FUNCTION_BLOCK XtsHardware_TestSuite
VAR
	nullHardware : XTSHardware('');
	MyXtsHardware : XTSHardware('') := (ExpectedNumberOfParts := 1, ExpectedNumberOfTracks := 1);
	localXpu: Xts_Library.I_TcIoXtsProcessingUnit;
	ThisTestSuite : TestSuite<TestSuiteParameter.MaxTestCount>('C:\ProgramData\Beckhoff\TwinCAT\3.1\Boot\XtsHardware_Tests.xml') := (TestSuiteName := 'XtsHardware Test Suite');
END_VAR

IF NOT MyXtsHardware.Initialised THEN
	MyXtsHardware.Initialise();
	RETURN;
END_IF

HardwareAcceptsTrackForDetection_Test();
HardwareAcceptsValidGetTrack_Test();
HardwareRejectsOnlyTrackRemove_Test();
HardwareIdentifiesNoXpu_Test();
HardwareRejectsCallsWithNoXPU_Test();
HardwareRejectsGetTrackWithHighTrackNum_Test();
HardwareRejectsGetTrackWithNull_Test();
HardwareRejectsHighIndexTrackRemoval_Test();
HardwareRejectsHighIndexTrackSet_Test();
HardwareRejectsNullTrackRemoval_Test();
HardwareRejectsNullTrackSet_Test();
HardwareReturnsCorrectMoverNumber_Test();
HardwareAcceptsValidMoverDetectionNumber_Test();
HardwareRejectsTooManyMoversForDetection_Test();
HardwareRejectsSetNegativeMoverNumber_Test();
HardwareWontCycleWithoutInit_Test();
RegisterXPU_Test();
HardwareAcceptsTriggerDetectionCommand_Test();
HardwareRejectsTriggerDetectionWithNoRef_Test();
HardwareAcceptsTriggerRedetectionCommand_Test();
HardwareRejectsTriggerRedetectionWithNoRef_Test();
HArdwareAcceptsMover1DetectionCommand_Test();
HardwareRejectsMover1DetectionInStandardMode_Test();

METHOD HArdwareAcceptsMover1DetectionCommand_Test
VAR_INST
	Expected : BOOL := TRUE;
	Actual	 : BOOL;
END_VAR
IF ThisTestSuite.Test(__POUNAME()).ExecuteTest() THEN
	localXpu.SetMoverIdDetectionMode(eMoverIdDetectionMode := MoverIdDetectionMode.Mover1);
	Actual := SUCCEEDED(MyXtsHardware.TriggerMoverIDDetection());
	ThisTestSuite.Test(__POUNAME()).AssertEqual(Expected, Actual);
END_IF
END_METHOD

METHOD HardwareAcceptsTrackForDetection_Test
VAR_INST
	Expected : BOOL := TRUE;
	Actual	 : BOOL;
END_VAR
IF ThisTestSuite.Test(__POUNAME()).ExecuteTest() THEN
	Actual := SUCCEEDED(MyXtsHardware.SetATrackForDetection(1));
	ThisTestSuite.Test(__POUNAME()).AssertEqual(Expected, Actual);
END_IF
END_METHOD

METHOD HardwareAcceptsTriggerDetectionCommand_Test
VAR_INST
	Expected : BOOL := TRUE;
	Actual	 : BOOL;
END_VAR
IF ThisTestSuite.Test(__POUNAME()).ExecuteTest() THEN
	Actual := SUCCEEDED(MyXtsHardware.TriggerMoverDetection());
	ThisTestSuite.Test(__POUNAME()).AssertEqual(Expected, Actual);
END_IF
END_METHOD

METHOD HardwareAcceptsTriggerRedetectionCommand_Test
VAR_INST
	Expected : BOOL := TRUE;
	Actual	 : BOOL;
END_VAR
IF ThisTestSuite.Test(__POUNAME()).ExecuteTest() THEN
	Actual := SUCCEEDED(MyXtsHardware.TriggerMoverRedetection());
	ThisTestSuite.Test(__POUNAME()).AssertEqual(Expected, Actual);
END_IF
END_METHOD

METHOD HardwareAcceptsValidGetTrack_Test
VAR_INST
	Expected : BOOL := TRUE;
	Actual	 : BOOL;
END_VAR
VAR
	temp: Xts_Library.I_XtsTrack;
END_VAR
IF ThisTestSuite.Test(__POUNAME()).ExecuteTest() THEN
	temp := MyXtsHardware.GetTrackInterfaceByNumber(1);
	Actual := temp <> 0;
	ThisTestSuite.Test(__POUNAME()).AssertEqual(Expected, Actual);
END_IF
END_METHOD

METHOD HardwareAcceptsValidMoverDetectionNumber_Test
VAR_INST
	Expected : BOOL := TRUE;
	Actual	 : BOOL;
END_VAR
IF ThisTestSuite.Test(__POUNAME()).ExecuteTest() THEN
	Actual := SUCCEEDED(MyXtsHardware.SetMoverNumberForDetection(2));
	ThisTestSuite.Test(__POUNAME()).AssertEqual(Expected, Actual);
END_IF
END_METHOD

METHOD HardwareIdentifiesNoXpu_Test : BOOL
VAR_INST
	Expected : BOOL := FALSE;
	Actual	 : BOOL;
END_VAR
IF ThisTestSuite.Test(__POUNAME()).ExecuteTest() THEN
	Actual := nullHardware.HasValidXPUReference();
	ThisTestSuite.Test(__POUNAME()).AssertEqual(Expected, Actual);
END_IF
END_METHOD

METHOD HardwareRejectsCallsWithNoXPU_Test : BOOL
VAR_INST
	Expected : BOOL := TRUE;
	Actual	 : BOOL;
END_VAR
IF ThisTestSuite.Test(__POUNAME()).ExecuteTest() THEN
	Actual := FAILED(nullHardware.Initialise());
	ThisTestSuite.Test(__POUNAME()).AssertEqual(Expected, Actual);
END_IF
END_METHOD

METHOD HardwareRejectsGetTrackWithHighTrackNum_Test
VAR_INST
	Expected : BOOL := TRUE;
	Actual	 : BOOL;
END_VAR
VAR
	temp: Xts_Library.I_XtsTrack;
END_VAR
IF ThisTestSuite.Test(__POUNAME()).ExecuteTest() THEN
	temp := MyXtsHardware.GetTrackInterfaceByNumber(3);
	Actual := temp = 0;
	ThisTestSuite.Test(__POUNAME()).AssertEqual(Expected, Actual);
END_IF
END_METHOD

METHOD HardwareRejectsGetTrackWithNull_Test
VAR_INST
	Expected : BOOL := TRUE;
	Actual	 : BOOL;
END_VAR
VAR
	temp: Xts_Library.I_XtsTrack;
END_VAR
IF ThisTestSuite.Test(__POUNAME()).ExecuteTest() THEN
	temp := MyXtsHardware.GetTrackInterfaceByNumber(0);
	Actual := temp = 0;
	ThisTestSuite.Test(__POUNAME()).AssertEqual(Expected, Actual);
END_IF
END_METHOD

METHOD HardwareRejectsHighIndexTrackRemoval_Test
VAR_INST
	Expected : BOOL := TRUE;
	Actual	 : BOOL;
END_VAR
IF ThisTestSuite.Test(__POUNAME()).ExecuteTest() THEN
	Actual := FAILED(MyXtsHardware.RemoveATrackFromDetection(3));
	ThisTestSuite.Test(__POUNAME()).AssertEqual(Expected, Actual);
END_IF
END_METHOD

METHOD HardwareRejectsHighIndexTrackSet_Test
VAR_INST
	Expected : BOOL := TRUE;
	Actual	 : BOOL;
END_VAR
IF ThisTestSuite.Test(__POUNAME()).ExecuteTest() THEN
	Actual := FAILED(MyXtsHardware.RemoveATrackFromDetection(3));
	ThisTestSuite.Test(__POUNAME()).AssertEqual(Expected, Actual);
END_IF
END_METHOD

METHOD HardwareRejectsMover1DetectionInStandardMode_Test
VAR_INST
	Expected : BOOL := TRUE;
	Actual	 : BOOL;
END_VAR
IF ThisTestSuite.Test(__POUNAME()).ExecuteTest() THEN
	localXpu.SetMoverIdDetectionMode(eMoverIdDetectionMode := MoverIdDetectionMode.Standard);
	Actual := FAILED(MyXtsHardware.TriggerMoverIDDetection());
	ThisTestSuite.Test(__POUNAME()).AssertEqual(Expected, Actual);
END_IF
END_METHOD

METHOD HardwareRejectsNullTrackRemoval_Test
VAR_INST
	Expected : BOOL := TRUE;
	Actual	 : BOOL;
END_VAR
IF ThisTestSuite.Test(__POUNAME()).ExecuteTest() THEN
	Actual := FAILED(MyXtsHardware.RemoveATrackFromDetection(0));
	ThisTestSuite.Test(__POUNAME()).AssertEqual(Expected, Actual);
END_IF
END_METHOD

METHOD HardwareRejectsNullTrackSet_Test
VAR_INST
	Expected : BOOL := TRUE;
	Actual	 : BOOL;
END_VAR
IF ThisTestSuite.Test(__POUNAME()).ExecuteTest() THEN
	Actual := FAILED(MyXtsHardware.SetATrackForDetection(0));
	ThisTestSuite.Test(__POUNAME()).AssertEqual(Expected, Actual);
END_IF
END_METHOD

METHOD HardwareRejectsOnlyTrackRemove_Test
VAR_INST
	Expected : BOOL := TRUE;
	Actual	 : BOOL;
END_VAR
IF ThisTestSuite.Test(__POUNAME()).ExecuteTest() THEN
	Actual := FAILED(MyXtsHardware.RemoveATrackFromDetection(1));
	ThisTestSuite.Test(__POUNAME()).AssertEqual(Expected, Actual);
END_IF
END_METHOD

METHOD HardwareRejectsSetNegativeMoverNumber_Test
VAR_INST
	Expected : BOOL := TRUE;
	Actual	 : BOOL;
END_VAR
IF ThisTestSuite.Test(__POUNAME()).ExecuteTest() THEN
	Actual := FAILED(MyXtsHardware.SetMoverNumberForDetection(-1));
	ThisTestSuite.Test(__POUNAME()).AssertEqual(Expected, Actual);
END_IF
END_METHOD

METHOD HardwareRejectsTooManyMoversForDetection_Test
VAR_INST
	Expected : BOOL := TRUE;
	Actual	 : BOOL;
END_VAR
IF ThisTestSuite.Test(__POUNAME()).ExecuteTest() THEN
	Actual := FAILED(MyXtsHardware.SetMoverNumberForDetection(20));
	ThisTestSuite.Test(__POUNAME()).AssertEqual(Expected, Actual);
END_IF
END_METHOD

METHOD HardwareRejectsTriggerDetectionWithNoRef_Test
VAR_INST
	Expected : BOOL := TRUE;
	Actual	 : BOOL;
END_VAR
IF ThisTestSuite.Test(__POUNAME()).ExecuteTest() THEN
	Actual := FAILED(nullHardware.TriggerMoverDetection());
	ThisTestSuite.Test(__POUNAME()).AssertEqual(Expected, Actual);
END_IF
END_METHOD

METHOD HardwareRejectsTriggerRedetectionWithNoRef_Test
VAR_INST
	Expected : BOOL := TRUE;
	Actual	 : BOOL;
END_VAR
IF ThisTestSuite.Test(__POUNAME()).ExecuteTest() THEN
	Actual := FAILED(nullHardware.TriggerMoverRedetection());
	ThisTestSuite.Test(__POUNAME()).AssertEqual(Expected, Actual);
END_IF
END_METHOD

METHOD HardwareReturnsCorrectMoverNumber_Test
VAR_INST
	Expected : BOOL := TRUE;
	Actual	 : BOOL;
END_VAR
IF ThisTestSuite.Test(__POUNAME()).ExecuteTest() THEN
	Actual := MyXtsHardware.GetNumberMoversDetected() = 5;
	ThisTestSuite.Test(__POUNAME()).AssertEqual(Expected, Actual);
END_IF
END_METHOD

METHOD HardwareWontCycleWithoutInit_Test : BOOL
VAR_INST
	Expected : BOOL := TRUE;
	Actual	 : BOOL;
END_VAR
IF ThisTestSuite.Test(__POUNAME()).ExecuteTest() THEN
	Actual := FAILED(nullHardware.Cycle());
	ThisTestSuite.Test(__POUNAME()).AssertEqual(Expected, Actual);
END_IF
END_METHOD

METHOD RegisterXPU_Test : BOOL
VAR_INST
	Expected : BOOL := TRUE;
	Actual	 : BOOL;
END_VAR
IF ThisTestSuite.Test(__POUNAME()).ExecuteTest() THEN
	Actual := MyXtsHardware.HasValidXPUReference();
	ThisTestSuite.Test(__POUNAME()).AssertEqual(Expected, Actual);
END_IF
END_METHOD

PROPERTY XPUInterface : I_TcIoXtsProcessingUnit
SET
localXpu := XPUInterface;
END_SET
END_PROPERTY

PROPERTY XtsHWInterface : I_TcIoXtsProcessingUnit
SET
MyXtsHardware.MyXpu :=  XtsHWInterface;
END_SET
END_PROPERTY

END_FUNCTION_BLOCK

(* stored: Version 1.1.0.1
   POU XtsHardware_TestSuite: Id {b560ca6a-e691-471a-a25d-3f29414ba80e}, SpecialFunc None
   Method HArdwareAcceptsMover1DetectionCommand_Test: Id {1eb9d286-88a2-4ceb-9442-caa77ceb3e4f}
   Method HardwareAcceptsTrackForDetection_Test: Id {fd2cec04-03de-4f58-93af-2288cf05eda1}
   Method HardwareAcceptsTriggerDetectionCommand_Test: Id {276c3e31-43f0-4f0a-ade3-22794a6bf2f4}
   Method HardwareAcceptsTriggerRedetectionCommand_Test: Id {4f7e235b-ae8d-420d-a721-1d686ea177fd}
   Method HardwareAcceptsValidGetTrack_Test: Id {0e46542d-c604-4447-8a3e-3ec02c688573}
   Method HardwareAcceptsValidMoverDetectionNumber_Test: Id {4c9fdbf0-8ba2-4715-a173-05b8e3911cd5}
   Method HardwareIdentifiesNoXpu_Test: Id {8917a178-edef-4eb2-9cd2-49d29f8c1ec8}
   Method HardwareRejectsCallsWithNoXPU_Test: Id {1788fe5c-f52a-4593-9903-c640bbecef8a}
   Method HardwareRejectsGetTrackWithHighTrackNum_Test: Id {68815c88-a416-44f3-8ffc-4330118a5ceb}
   Method HardwareRejectsGetTrackWithNull_Test: Id {e99ddcf3-f9fa-4666-9905-b72e0c37553c}
   Method HardwareRejectsHighIndexTrackRemoval_Test: Id {37d87a5b-ee31-480d-aa9a-95e920fc471d}
   Method HardwareRejectsHighIndexTrackSet_Test: Id {853c738b-2619-467e-9ed0-169bb122a5bc}
   Method HardwareRejectsMover1DetectionInStandardMode_Test: Id {7262a4cd-1e5d-4acb-8d51-66ab87154709}
   Method HardwareRejectsNullTrackRemoval_Test: Id {372f9c0b-9be7-4c16-90ad-79978c12fc6c}
   Method HardwareRejectsNullTrackSet_Test: Id {27465936-dd7b-4282-8d76-6b5f2d21fe9b}
   Method HardwareRejectsOnlyTrackRemove_Test: Id {3c4edcdb-2ae4-4b9c-bfd7-ab42758989a3}
   Method HardwareRejectsSetNegativeMoverNumber_Test: Id {1b71a8a8-e8c5-44e1-9189-d9e60ce551cf}
   Method HardwareRejectsTooManyMoversForDetection_Test: Id {2e4a8332-8580-4d8c-aa0e-f65bc25da910}
   Method HardwareRejectsTriggerDetectionWithNoRef_Test: Id {9ed3090f-a74b-4abf-aa18-8a65a899d503}
   Method HardwareRejectsTriggerRedetectionWithNoRef_Test: Id {51d9dbf1-3bde-4d89-94eb-76b62afc1775}
   Method HardwareReturnsCorrectMoverNumber_Test: Id {a5ce0842-b23f-4b90-95c8-5e791ebcc2dd}
   Method HardwareWontCycleWithoutInit_Test: Id {fba77493-9432-4925-a6b5-53c91b6f648a}
   Method RegisterXPU_Test: Id {b248b030-f2bc-411a-8466-8dc5754b8803}
   Property XPUInterface: Id {87d6f6c6-5136-44e2-ac7b-65ad1ff46c0c}
   Set Set: Id {e4d6cd76-f880-4b01-bc99-1cd1f9d86c90}
   Property XtsHWInterface: Id {63a37f49-ad64-4614-b378-51dbfb998d3f}
   Set Set: Id {4ea51632-817b-4a8b-8fcb-d193cdb7f393} *)
